FUNCTION_BLOCK FB_System
VAR_INPUT
	bEtwas		: BOOL;
END_VAR
VAR_OUTPUT
	bError		: BOOL;
	bReady		: BOOL;
END_VAR
VAR
END_VAR

END_FUNCTION_BLOCK

(* stored: Version 1.1.0.1, ProductVersion 3.1.4024.12
   POU FB_System: Id {5b40ff5c-73f8-4fe6-a7ad-41d6ddec4ec6}, SpecialFunc None *)
